{attribute 'pack_mode' := '1'}
    {attribute 'OPC.UA.DA' := '1'}
    {attribute 'OPC.UA.DA.StructuredType' := '1'}
    (*
    ST_RW_Plc_Info_S71200_HMI_IgnitionExp
    ==================================================
    Generated from Ignition UDT: RW_PLC_Info_S71200
    Total tags: 12
    Generated on: 2025-09-16 15:04:58
    *)
    TYPE ST_RW_Plc_Info_S71200_HMI_IgnitionExp :
    STRUCT
        {attribute 'OPC.UA.DA' := '1'}
        {attribute 'OPC.UA.DA.Access' := '1'}
        KW_Device_ScanRateMs : DINT := 0;		// Read-only tag
        {attribute 'OPC.UA.DA' := '1'}
        {attribute 'OPC.UA.DA.Access' := '1'}
        KW_Device_SuccessfulReads : SINT := 0;		// Read-only tag
        {attribute 'OPC.UA.DA' := '1'}
        {attribute 'OPC.UA.DA.Access' := '1'}
        KW_Device_Error : BOOL := FALSE;		// Read-only tag
        {attribute 'OPC.UA.DA' := '1'}
        {attribute 'OPC.UA.DA.Access' := '1'}
        KW_Device_SuccessfulWrites : SINT := 0;		// Read-only tag
        {attribute 'OPC.UA.DA' := '1'}
        {attribute 'OPC.UA.DA.Access' := '1'}
        KW_Device_Description : STRING := '';		// Read-only tag

        {attribute 'OPC.UA.DA' := '1'}
        {attribute 'OPC.UA.DA.Access' := '1'}
        KW_Device_ScanMode : STRING := '';		// Read-only tag
        {attribute 'OPC.UA.DA' := '1'}
        KW_ForceSymbolReload : BOOL := FALSE;
        {attribute 'OPC.UA.DA' := '1'}
        {attribute 'OPC.UA.DA.Access' := '1'}
        KW_Device_Enabled : BOOL := FALSE;		// Read-only tag
        {attribute 'OPC.UA.DA' := '1'}
        {attribute 'OPC.UA.DA.Access' := '1'}
        KW_Device_SecondsInError : SINT := 0;		// Read-only tag
        {attribute 'OPC.UA.DA' := '1'}
        {attribute 'OPC.UA.DA.Access' := '1'}
        KW_Device_FailedReads : SINT := 0;		// Read-only tag

        {attribute 'OPC.UA.DA' := '1'}
        {attribute 'OPC.UA.DA.Access' := '1'}
        KW_Device_ActiveTagCount : DINT := 0;		// Read-only tag
        {attribute 'OPC.UA.DA' := '1'}
        {attribute 'OPC.UA.DA.Access' := '1'}
        KW_Device_FailedWrites : SINT := 0;		// Read-only tag
    END_STRUCT
    END_TYPE

(* stored: Version 1.1.0.1
   DUT ST_RW_Plc_Info_S71200_HMI_IgnitionExp: Id {7a03bb4c-f681-4bde-8ed9-d99fed5d9fe9} *)
